// TIA Portal V17 export
// export: Created 2021-12-03T08:13:07.8619751Z, ExportSetting WithDefaults, DisplayName Totally Integrated Automation Portal, DisplayVersion V17, DisplayName TIA Portal Openness, DisplayVersion V17, DisplayName TIA Portal Version Control Interface, DisplayVersion V17, DisplayName STEP 7 Professional, DisplayVersion V17, DisplayName STEP 7 Safety, DisplayVersion V17, DisplayName WinCC Advanced, DisplayVersion V17
FUNCTION "FC_SignCtrl" : Void   // FC800, FBD
VERSION : 0.1
// stored: AutoNumber false, IsIECCheckEnabled false, UDAEnableTagReadback false
   VAR_INPUT
      I_LmpTst : Bool;   // 1=Lamp Test (Highest Priority)
      I_LmpMd1 : Bool;   // Mode 1 (High Priority)
      I_LmpMd1Clk : Bool;   // Mode 1 (Clock)
      I_LmpMd2 : Bool;   // Mode 2 (Middle Priority)
      I_LmpMd2Clk : Bool;   // Mode 2 (Clock)
      I_LmpMd3 : Bool;   // Mode 3 (Low Priority)
      I_LmpMd3Clk : Bool;   // Mode 3 (Clock)
   END_VAR
   VAR_OUTPUT
      O_Lmp : Bool;   // Lamp
   END_VAR
BEGIN

REGION Network 1: Functional Description
   // This FC controlled the output depends on the input and is used for controlling lamps.
   // If more than one input is active the output will controlled by the input which have the higher priority.
   // There are 4 modes...
   // Mode 1: I_LmpTst highest priority
   // Mode 2: I_ LmpMd1 high priority
   // Mode 3: I_ LmpMd2 low priority
   // Mode 4: I_LmpMd3 lowest priority
   // The inputs I_LmpMd1Clk, I_LmpMd2Clk, I_LmpMd3Clk, is the clock signal of the several inputs.
END_REGION

REGION Network 2: Lamp Test
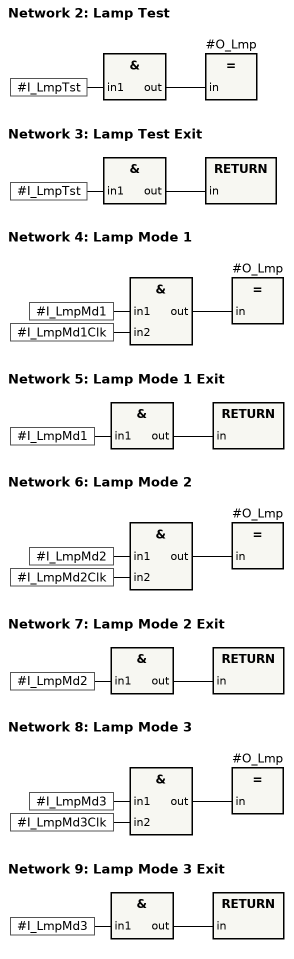
   #O_Lmp := #I_LmpTst;
END_REGION

REGION Network 3: Lamp Test Exit
   IF #I_LmpTst THEN
       ENO := TRUE;
       RETURN;
   END_IF;
END_REGION

REGION Network 4: Lamp Mode 1
   #O_Lmp := #I_LmpMd1 AND #I_LmpMd1Clk;
END_REGION

REGION Network 5: Lamp Mode 1 Exit
   IF #I_LmpMd1 THEN
       ENO := TRUE;
       RETURN;
   END_IF;
END_REGION

REGION Network 6: Lamp Mode 2
   #O_Lmp := #I_LmpMd2 AND #I_LmpMd2Clk;
END_REGION

REGION Network 7: Lamp Mode 2 Exit
   IF #I_LmpMd2 THEN
       ENO := TRUE;
       RETURN;
   END_IF;
END_REGION

REGION Network 8: Lamp Mode 3
   #O_Lmp := #I_LmpMd3 AND #I_LmpMd3Clk;
END_REGION

REGION Network 9: Lamp Mode 3 Exit
   IF #I_LmpMd3 THEN
       ENO := TRUE;
       RETURN;
   END_IF;
END_REGION

REGION Network 10: Block End
END_REGION
END_FUNCTION
